PROGRAM DoorControlLogic
VAR
	{attribute 'OPC.UA.DA' := '1'}	
	chart_cssd_door_Status						:	BOOL;	// Status of door contact - True:Open | False:Close
	
	{attribute 'OPC.UA.DA' := '1'}	
	chart_cssd_door_Open_Command	AT %I*		: 	BOOL;	// Open Door 1 command from robot

	{attribute 'OPC.UA.DA' := '1'}			
	chart_cssd_door_Close_Command	AT %I*		:	BOOL	:= FALSE;	// Close Door 1 command from robot, init to be false

	{attribute 'OPC.UA.DA' := '1'}		
	chart_cssd_door_Opened_Signal	AT %I*		:	BOOL;
	
	{attribute 'OPC.UA.DA' := '1'}		
	chart_cssd_door_Closed_Signal	AT %I*		: 	BOOL;
	
	{attribute 'OPC.UA.DA' := '1'}		
	chart_cssd_door_Hold			AT %Q*		: 	BOOL;
	
	chart_cssd_door_Contact			AT %Q* 		: 	BOOL	:= FALSE;	// Output to close door contact, init to be false
	
END_VAR

IF chart_cssd_door_Close_Command = TRUE AND NOT chart_cssd_door_Open_Command = TRUE THEN
	chart_cssd_door_Contact := FALSE;
	chart_cssd_door_Hold := FALSE; 
	ELSIF chart_cssd_door_Open_Command = TRUE AND chart_cssd_door_Close_Command = FALSE THEN
		chart_cssd_door_Contact := TRUE;
		chart_cssd_door_Hold := TRUE;		
		ELSIF chart_cssd_door_Open_Command = TRUE AND chart_cssd_door_Close_Command = TRUE THEN
			chart_cssd_door_Contact := FALSE;
			chart_cssd_door_Hold := FALSE;
			chart_cssd_door_Open_Command := FALSE;
			ELSIF chart_cssd_door_Open_Command := FALSE AND chart_cssd_door_Close_Command = FALSE THEN
				chart_cssd_door_Contact := FALSE;
				chart_cssd_door_Hold := FALSE;
				chart_cssd_door_Open_Command := FALSE;
//			ELSIF chart_cssd_door_Open_Command := FALSE AND chart_cssd_door_Close_Command = TRUE THEN
//				chart_cssd_door_Contact := TRUE;
//				chart_cssd_door_Hold := TRUE;
//				chart_cssd_door_Open_Command := TRUE; Commented out as conditions are the same as first condition
	END_IF

IF chart_cssd_door_Opened_Signal = TRUE AND chart_cssd_door_Closed_Signal = FALSE THEN
	chart_cssd_door_Status := TRUE;
	ELSIF chart_cssd_door_Closed_Signal = TRUE AND chart_cssd_door_Opened_Signal = FALSE THEN
		chart_cssd_door_Status := FALSE;
		ELSE
			chart_cssd_door_Status := FALSE;
	END_IF

END_PROGRAM

(* stored: Version 1.1.0.1, ProductVersion 3.1.4022.18
   POU DoorControlLogic: Id {5d89914e-5fc5-4bf5-a467-154940aa51ec}, SpecialFunc None *)
